Fanuc KAREL source: kt00130.KL

PROGRAM KT00130
%STACKSIZE=65535
%PRIORITY=65535
%NOLOCKGROUP
VAR
I1 : INTEGER
I2 : INTEGER
OUT : REAL
BEGIN
I1=2
I2=3
I1=2
I2=3
OUT=(I1 DIV I2)
END KT00130
